// SIMATIC S7-200 project (STEP 7-Micro/WIN), CPU 221 REL 01.10

SYMBOL_TABLE USER1
start            I0.0     // khoi dong he thong
estop            I0.1     // dung he thong
cb1              I0.2     // cam bien phat hien xe vao
cb2              I0.3     // cam bien phat hien xe ra
cb3              I0.4     // cong tac hanh trinh gioi han nang barie cua vao
cb4              I0.5     // cong tac hanh trinh giai han ha barie cua vao
cb5              I0.6     // cong tac hanh trinh gioi han nang barie cua ra
cb6              I0.7     // cong tac hanh trinh gioi han ha barie cua ra
M1T              Q0.0     // dong co barie mo cua vao
M1N              Q0.1     // dong co barie dong cua vao
M2T              Q0.2     // dong co barie mo cua ra
M2N              Q0.3     // dong co barie dong cua ra
Den              Q0.4     // den bao day xe
END_SYMBOL_TABLE

ORGANIZATION_BLOCK MAIN:OB1
TITLE=PROGRAM COMMENTS
BEGIN
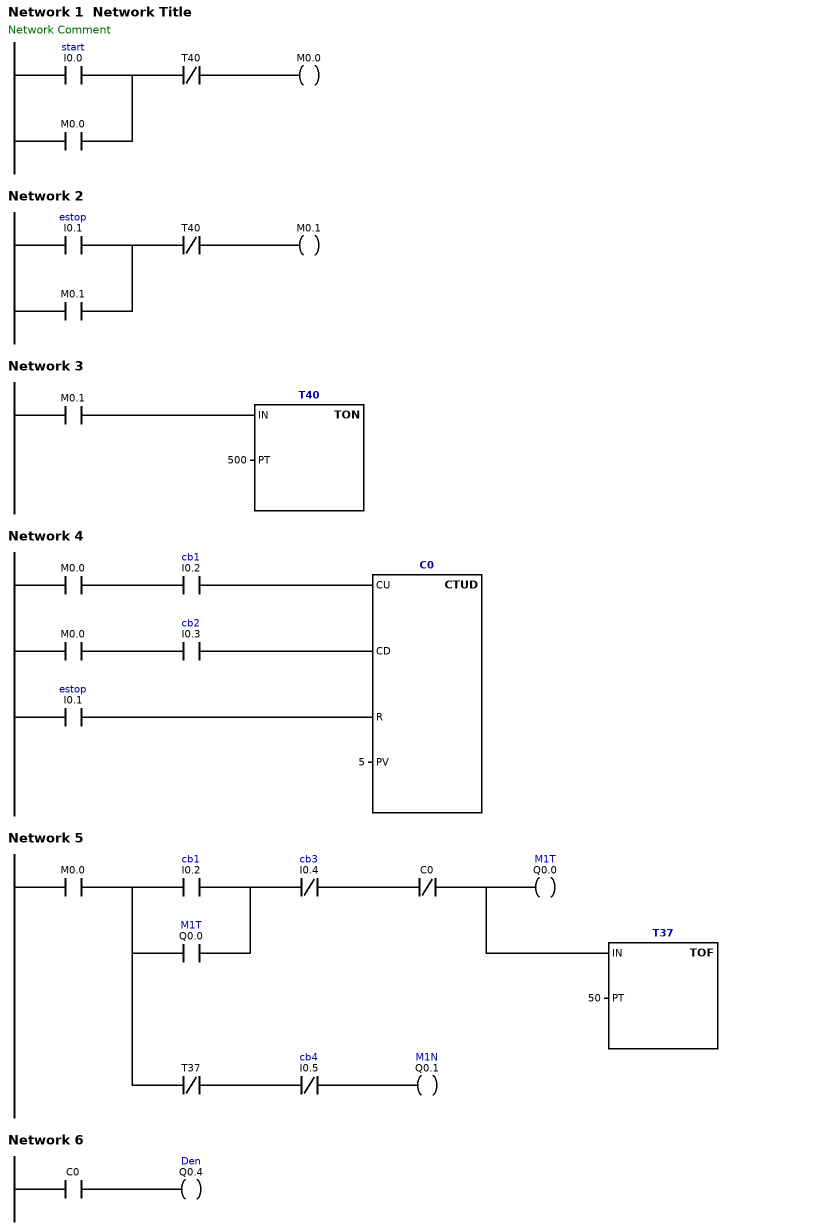
Network 1 // Network Title
// Network Comment
LD     start:I0.0
O      M0.0
AN     T40
=      M0.0
Network 2
LD     estop:I0.1
O      M0.1
AN     T40
=      M0.1
Network 3
LD     M0.1
TON    T40, 500
Network 4
LD     M0.0
A      cb1:I0.2
LD     M0.0
A      cb2:I0.3
LD     estop:I0.1
CTUD   C0, 5
Network 5
LD     M0.0
LPS
LD     cb1:I0.2
O      M1T:Q0.0
AN     cb3:I0.4
AN     C0
ALD
=      M1T:Q0.0
TOF    T37, 50
LPP
AN     T37
AN     cb4:I0.5
=      M1N:Q0.1
Network 6
LD     C0
=      Den:Q0.4
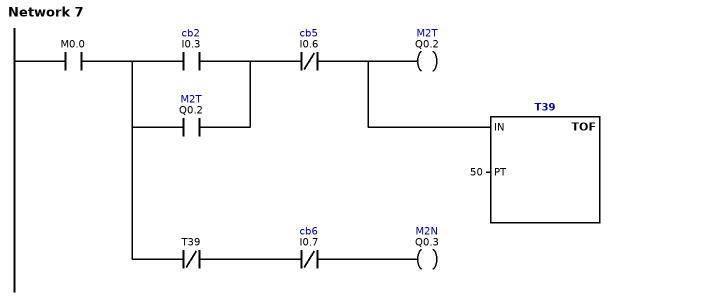
Network 7
LD     M0.0
LPS
LD     cb2:I0.3
O      M2T:Q0.2
AN     cb5:I0.6
ALD
=      M2T:Q0.2
TOF    T39, 50
LPP
AN     T39
AN     cb6:I0.7
=      M2N:Q0.3
END_ORGANIZATION_BLOCK
